// TIA Portal project "Registerlager" (V14)

(* hardware
DEVICE "S71500/ET200MP-Station_1"  S7-1500 station
   slot 0: "Profilschiene_0"  Rack  6ES7 590-1***0-0AA0
   slot 1: "PLC_1"  CPU 1512C-1 PN  6ES7 512-1CK00-0AB0  V2.1
      slot 3: "CPU-Display_1"  6ES7591-1AA00-0AA0
DEVICE "HMI_1"  TP700 Comfort
   slot 0: "TP700 Comfort"  TP700 Comfort  6AV2 124-0GC01-0AX0  14.0.1.0
   slot 1: "HMI_RT_1"  TP700 Comfort  6AV2 124-0GC01-0AX0  14.0.1.0
   slot 5: "HMI_1.IE_CP_1"  PROFINET Interface  14.0.1.0
      slot 1: "PROFINET Schnittstelle_1"  PROFINET Interface
         slot 1: "Port_1"  Port
         slot 2: "Port_2"  Port
   slot 7: "HMI_1.MPI/DP_CP_1"  MPI/DP Interface  14.0.1.0
*)

// ===== PLC "PLC_1"  CPU 1512C-1 PN =====
// protected blocks, not shown: "Anzeigeelemente HMI", "Bedienelemente HMI", "Bedienung HMI"

VAR_GLOBAL   // PLC tag table "Standard-Variablentabelle"
   "CHAIN_REGISTER" AT %I10.0 : Bool;   // Förderkette Registerlager, Reed-Kontakt Schließer
   "REGISTER_ENGAGED" AT %I10.1 : Bool;   // Registerlager belegt, Optokoppler Öffner
   "BELT_ENGAGED" AT %I10.2 : Bool;   // Förderband belegt, Näherungsschalter Schließer
   "READ_SENSOR1" AT %I10.3 : Bool;   // Lesestation Sensor 1, Reed-Kontakt Schließer
   "READ_SENSOR2" AT %I10.4 : Bool;   // Lesestation Sensor 2, Reed-Kontakt Schließer
   "CONTROL_KEY" AT %I10.5 : Bool;   // Bedientaster, Schließer
   "CHAIN_ON" AT %Q4.0 : Bool;   // Förderkette Registerlager an
   "BELT_ON" AT %Q4.1 : Bool;   // Förderband an
   "LED_ON" AT %Q4.2 : Bool;   // LED an
   "BOX_NO" AT %MD1000 : DInt;   // Nummer der Box auf dem Förderband
   "SPS_ENABLE" AT %M1004.0 : Bool;   // Bedienung der Aktoren per Programm
   "CONTROL_KEY_HMI" AT %M1004.1 : Bool;   // Bedientaster (HMI)
   "RESET" AT %E11.7 : Bool;   // Taster zur freien Verfügung, Schließer
   "Merker, 15 sec timer done" AT %M0.1 : Bool;
   "Tag_1" AT %M0.2 : Bool;
   "Merker TOF aktiv" AT %M0.0 : Bool;
   "Tag_2" AT %M0.3 : Bool;
   "BOX_COUNTER_BOTH" AT %MW3 : Int;
   "BOX_COUNTER1" AT %MW6 : Int;
   "BOX_COUNTER2" AT %MW8 : Int;
   "Tag_3" AT %M0.4 : Bool;
   "Tag_4" AT %M0.5 : Bool;
END_VAR

// folder: System blocks/Program resources

DATA_BLOCK "IEC_Timer_0_DB_1"   // DB2
{ S7_Optimized_Access := 'TRUE' }
AUTHOR : Simatic
FAMILY : IEC
NAME : IEC_TMR
VERSION : 1.0
// stored: InstanceOfName IEC_TIMER
"IEC_TIMER"
BEGIN
END_DATA_BLOCK

DATA_BLOCK "IEC_Counter_0_DB"   // DB3
{ S7_Optimized_Access := 'TRUE' }
AUTHOR : Simatic
FAMILY : IEC
NAME : CNTR
VERSION : 1.0
// stored: InstanceOfName IEC_COUNTER
"IEC_COUNTER"
BEGIN
END_DATA_BLOCK

DATA_BLOCK "IEC_Counter_1_DB"   // DB4
{ S7_Optimized_Access := 'TRUE' }
AUTHOR : Simatic
FAMILY : IEC
NAME : CNTR
VERSION : 1.0
// stored: InstanceOfName IEC_COUNTER
"IEC_COUNTER"
BEGIN
END_DATA_BLOCK

// folder: (top level)

ORGANIZATION_BLOCK "Main"   // OB1, FBD, ProgramCycle
TITLE = "Main Program Sweep (Cycle)"
{ S7_Optimized_Access := 'TRUE' }
VERSION : 0.1
   VAR_INPUT
      Initial_Call : Bool;   // Initial call of this OB
      Remanence : Bool;   // =True, if remanent data are available
   END_VAR
   VAR_TEMP   // added for the SCL form of the ladder/FBD networks
      _w1 : Bool;
      _w2 : Bool;
   END_VAR
BEGIN

REGION Network 1: Förderband an
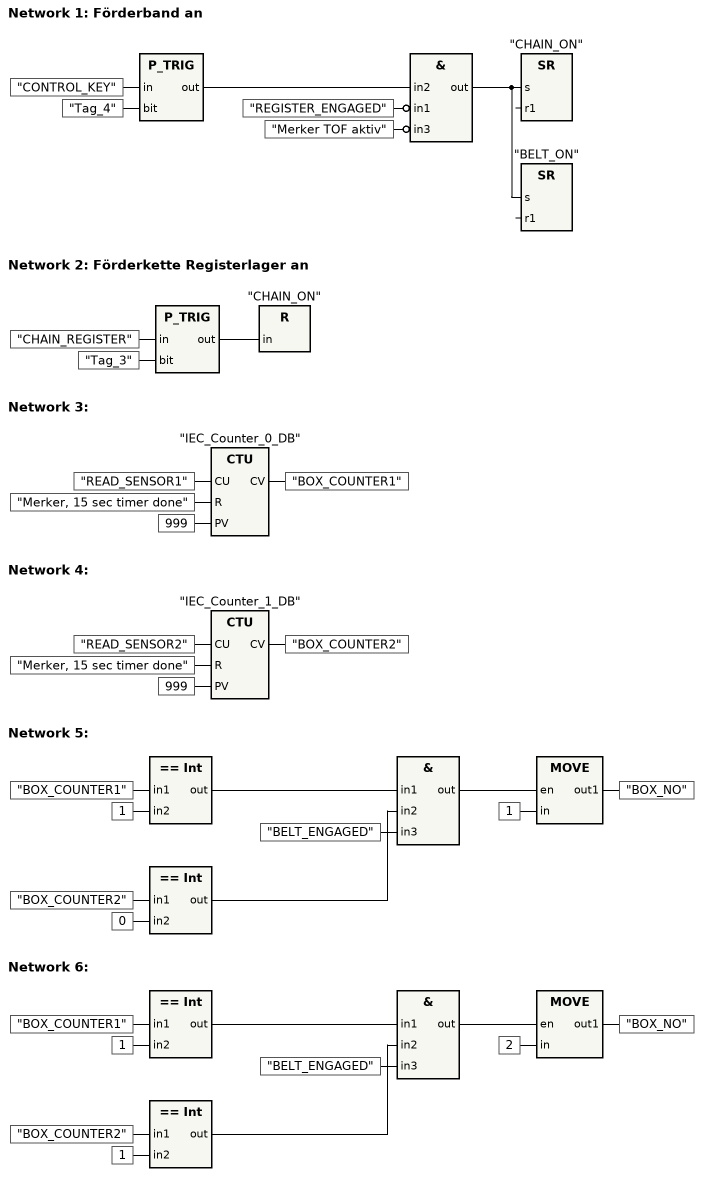
   #_w1 := "CONTROL_KEY" AND NOT "Tag_4";   // rising edge
   "Tag_4" := "CONTROL_KEY";
   #_w2 := #_w1 AND NOT "REGISTER_ENGAGED" AND NOT "Merker TOF aktiv";
   IF #_w2 THEN
       "CHAIN_ON" := TRUE;   // SR flip-flop
       "BELT_ON" := TRUE;   // SR flip-flop
   END_IF;
END_REGION

REGION Network 2: Förderkette Registerlager an
   #_w1 := "CHAIN_REGISTER" AND NOT "Tag_3";   // rising edge
   "Tag_3" := "CHAIN_REGISTER";
   IF #_w1 THEN "CHAIN_ON" := FALSE; END_IF;
END_REGION

REGION Network 3
   "IEC_Counter_0_DB".CTU(CU := "READ_SENSOR1",
                          R := "Merker, 15 sec timer done",
                          PV := 999,
                          CV => "BOX_COUNTER1");
END_REGION

REGION Network 4
   "IEC_Counter_1_DB".CTU(CU := "READ_SENSOR2",
                          R := "Merker, 15 sec timer done",
                          PV := 999,
                          CV => "BOX_COUNTER2");
END_REGION

REGION Network 5
   IF ("BOX_COUNTER1" = 1) AND ("BOX_COUNTER2" = 0) AND "BELT_ENGAGED" THEN "BOX_NO" := 1; END_IF;
END_REGION

REGION Network 6
   IF ("BOX_COUNTER1" = 1) AND ("BOX_COUNTER2" = 1) AND "BELT_ENGAGED" THEN "BOX_NO" := 2; END_IF;
END_REGION

REGION Network 7
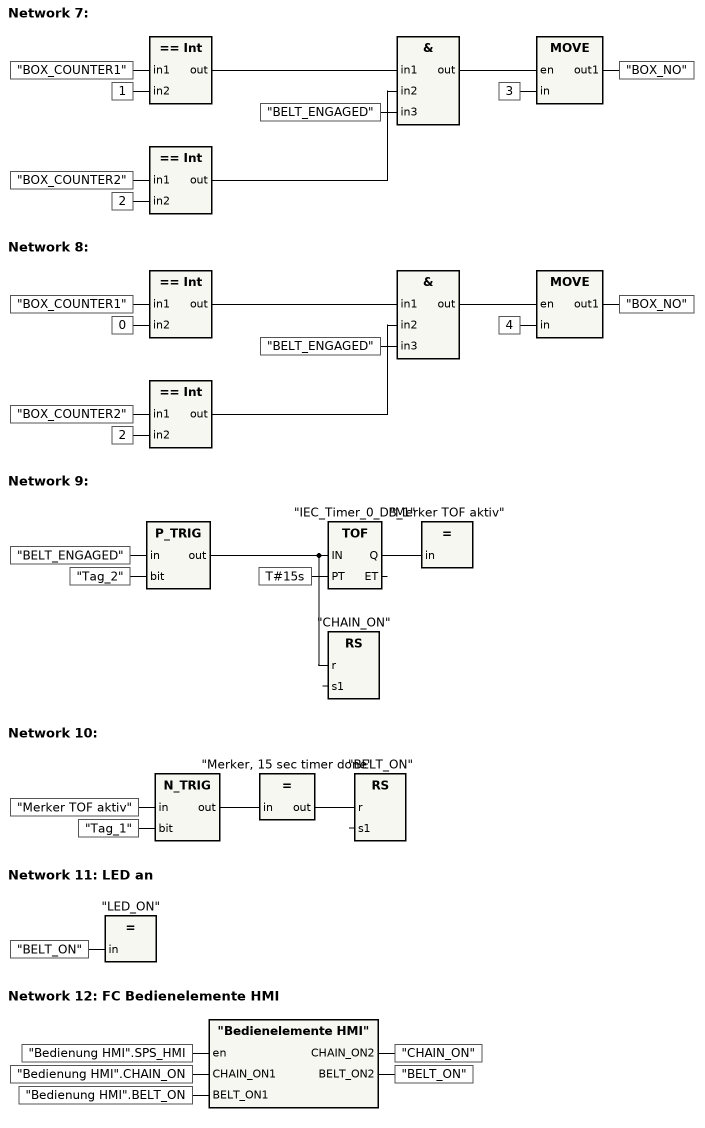
   IF ("BOX_COUNTER1" = 1) AND ("BOX_COUNTER2" = 2) AND "BELT_ENGAGED" THEN "BOX_NO" := 3; END_IF;
END_REGION

REGION Network 8
   IF ("BOX_COUNTER1" = 0) AND ("BOX_COUNTER2" = 2) AND "BELT_ENGAGED" THEN "BOX_NO" := 4; END_IF;
END_REGION

REGION Network 9
   #_w1 := "BELT_ENGAGED" AND NOT "Tag_2";   // rising edge
   "Tag_2" := "BELT_ENGAGED";
   "IEC_Timer_0_DB_1".TOF(IN := #_w1, PT := T#15s);
   "Merker TOF aktiv" := "IEC_Timer_0_DB_1".Q;
   IF #_w1 THEN
       "CHAIN_ON" := FALSE;   // RS flip-flop
   END_IF;
END_REGION

REGION Network 10
   #_w1 := NOT "Merker TOF aktiv" AND "Tag_1";   // falling edge
   "Tag_1" := "Merker TOF aktiv";
   "Merker, 15 sec timer done" := #_w1;
   IF #_w1 THEN
       "BELT_ON" := FALSE;   // RS flip-flop
   END_IF;
END_REGION

REGION Network 11: LED an
   "LED_ON" := "BELT_ON";
END_REGION

REGION Network 12: FC Bedienelemente HMI
   IF "Bedienung HMI".SPS_HMI THEN
       "Bedienelemente HMI"(CHAIN_ON1 := "Bedienung HMI".CHAIN_ON,
                            BELT_ON1 := "Bedienung HMI".BELT_ON,
                            CHAIN_ON2 => "CHAIN_ON",
                            BELT_ON2 => "BELT_ON");
   END_IF;
END_REGION

REGION Network 13: FC Anzeigeelemente HMI
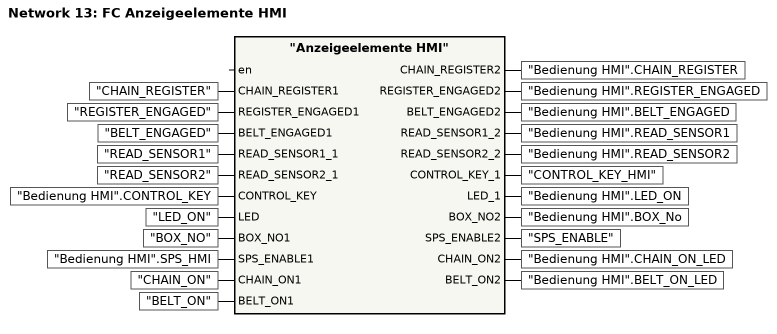
   "Anzeigeelemente HMI"(CHAIN_REGISTER1 := "CHAIN_REGISTER",
                         REGISTER_ENGAGED1 := "REGISTER_ENGAGED",
                         BELT_ENGAGED1 := "BELT_ENGAGED",
                         READ_SENSOR1_1 := "READ_SENSOR1",
                         READ_SENSOR2_1 := "READ_SENSOR2",
                         CONTROL_KEY := "Bedienung HMI".CONTROL_KEY,
                         LED := "LED_ON",
                         BOX_NO1 := "BOX_NO",
                         SPS_ENABLE1 := "Bedienung HMI".SPS_HMI,
                         CHAIN_ON1 := "CHAIN_ON",
                         BELT_ON1 := "BELT_ON",
                         CHAIN_REGISTER2 => "Bedienung HMI".CHAIN_REGISTER,
                         REGISTER_ENGAGED2 => "Bedienung HMI".REGISTER_ENGAGED,
                         BELT_ENGAGED2 => "Bedienung HMI".BELT_ENGAGED,
                         READ_SENSOR1_2 => "Bedienung HMI".READ_SENSOR1,
                         READ_SENSOR2_2 => "Bedienung HMI".READ_SENSOR2,
                         CONTROL_KEY_1 => "CONTROL_KEY_HMI",
                         LED_1 => "Bedienung HMI".LED_ON,
                         BOX_NO2 => "Bedienung HMI".BOX_No,
                         SPS_ENABLE2 => "SPS_ENABLE",
                         CHAIN_ON2 => "Bedienung HMI".CHAIN_ON_LED,
                         BELT_ON2 => "Bedienung HMI".BELT_ON_LED);
END_REGION
END_ORGANIZATION_BLOCK

(* ===== HMI "HMI_RT_1" =====
system functions are stored by id; their names below are inferred from use
connection "HMI_Verbindung_1": ETHERNET, S7_1500_OMS

HMI tags "Standard-Variablentabelle"
   "Bedienung HMI_CHAIN_REGISTER" : Bool = PLC "Bedienung HMI".CHAIN_REGISTER, 1 s
   "Bedienung HMI_REGISTER_ENGAGED" : Bool = PLC "Bedienung HMI".REGISTER_ENGAGED, 1 s
   "Bedienung HMI_BELT_ENGAGED" : Bool = PLC "Bedienung HMI".BELT_ENGAGED, 1 s
   "Bedienung HMI_READ_SENSOR1" : Bool = PLC "Bedienung HMI".READ_SENSOR1, 1 s
   "Bedienung HMI_READ_SENSOR2" : Bool = PLC "Bedienung HMI".READ_SENSOR2, 1 s
   "Bedienung HMI_CONTROL_KEY" : Bool = PLC "Bedienung HMI".CONTROL_KEY, 1 s
   "Bedienung HMI_CHAIN_ON" : Bool = PLC "Bedienung HMI".CHAIN_ON, 1 s
   "Bedienung HMI_BELT_ON" : Bool = PLC "Bedienung HMI".BELT_ON, 1 s
   "Bedienung HMI_LED_ON" : Bool = PLC "Bedienung HMI".LED_ON, 1 s
   "Bedienung HMI_BOX_No" : Int = PLC "Bedienung HMI".BOX_No AT %DB1.DBX0.0, 1 s
   "Bedienung HMI_SPS_HMI" : Bool = PLC "Bedienung HMI".SPS_HMI AT %DB1.DBX0.0, 1 s
   "Bedienung HMI_CHAIN_ON_LED" : Bool = PLC "Bedienung HMI".CHAIN_ON_LED AT %DB1.DBX0.0, 1 s
   "Bedienung HMI_BELT_ON_LED" : Bool = PLC "Bedienung HMI".BELT_ON_LED AT %DB1.DBX0.0, 1 s

text list "Textliste_Bildnamen": 1 'Grundbild'; 2 'Systembilder'; 3 'SIMATIC PLC Systemdiagnose'

screen "Bild_1" 800x480
   Button "Schaltfläche_1" at 304,60 size 152x42; TextOff 'Bedientaste'
      on Press: SetTag("Bedienung HMI_CONTROL_KEY", 1)
      on Release: ResetBit("Bedienung HMI_CONTROL_KEY")
   Button "Schaltfläche_2" at 170,385 size 153x40; TextOff 'Förderkette'
      on Press: SetTag("Bedienung HMI_CHAIN_ON", 1)
      on Release: ResetBit("Bedienung HMI_CHAIN_ON")
   Button "Schaltfläche_3" at 429,385 size 153x40; TextOff 'Förderband'
      on Press: SetTag("Bedienung HMI_BELT_ON", 1)
      on Release: ResetBit("Bedienung HMI_BELT_ON")
   Circle "Kreis_2" at 487,60 size 43x43
      Visibility <- "Bedienung HMI_LED_ON"
   TextField "Textfeld_1" at 199,182 size 83x23; Text 'Sensor 1'
   TextField "Textfeld_2" at 435,180 size 83x23; Text 'Sensor 2'
   TextField "Textfeld_3" at 578,60 size 77x43; Text 'BOX'
   IOField "EA-Feld_1" at 675,41 size 51x83; FormatPattern 9
      ProcessValue <- "Bedienung HMI_BOX_No"
   Circle "Kreis_5" at 539,172 size 43x43
      Visibility <- "Bedienung HMI_READ_SENSOR2"
   Circle "Kreis_6" at 292,172 size 43x43
      Visibility <- "Bedienung HMI_READ_SENSOR1"
   Circle "Kreis_8" at 404,280 size 43x43
      Visibility <- "Bedienung HMI_BELT_ENGAGED"
   TextField "Textfeld_4" at 310,287 size 90x23; Text 'Fb belegt'
   Circle "Kreis_10" at 229,280 size 43x43
      Visibility <- "Bedienung HMI_REGISTER_ENGAGED"
   TextField "Textfeld_5" at 81,287 size 146x23; Text 'Register belegt'
   TextField "Textfeld_6" at 491,287 size 180x23; Text 'Sensor Förderkette'
   Circle "Kreis_12" at 672,279 size 43x43
      Visibility <- "Bedienung HMI_CHAIN_REGISTER"
   Circle "Kreis_14" at 93,382 size 43x43
      Visibility <- "Bedienung HMI_CHAIN_ON_LED"
   Circle "Kreis_16" at 624,382 size 43x43
      Visibility <- "Bedienung HMI_BELT_ON_LED"
   Switch "Schalter_1" at 69,36 size 120x67; CaptionText 'Switch'; TextOff 'SPS'; TextOn 'HMI'
      ProcessValue <- "Bedienung HMI_SPS_HMI"
*)